FUNCTION_BLOCK FB_Blinker1
VAR_INPUT
	bStart: BOOL;         	//Start signal 
	tSignalTimeOn: TIME;  	//Pulse Time On
	tSignalTimeOff: TIME;	//Pulse Time Off
END_VAR
VAR_OUTPUT
	bOut: BOOL;				//Output pulse 
END_VAR
VAR
	fbTimerA: TON;			//TimerA Initialization
	fbTimerB: TON;			//TimerB Initialization
END_VAR

// Timer A Parameterization
fbTimerA(IN := (bStart AND NOT fbTimerB.Q),
		PT := tSignalTimeOn,
		Q => bOut
		);

// Timer B Parameterization	
fbTimerB(IN := fbTimerA.Q,
		PT := tSignalTimeOff,
		);

END_FUNCTION_BLOCK

(* stored: Version 1.1.0.1, ProductVersion 3.1.4024.4
   POU FB_Blinker1: Id {493f8cd2-7c29-4cac-9141-4d447a048dbe}, SpecialFunc None *)
